(* IEC 61131-3 sources: plc_path_sender/, 1 file *)

(* ---- A1_Input_Normalizer.st ---- *)
(*****************************************************
 A1 Input Normalizer - ST Program Skeleton
 Purpose: Provide structure only; logic intentionally omitted.
*****************************************************)

PROGRAM A1_Input_Normalizer
VAR
    (* === Inputs from upstream sources === *)
    RawInput_1 : INT; (* Placeholder for raw input channel 1 *)
    RawInput_2 : INT; (* Placeholder for raw input channel 2 *)

    (* === Configuration / tuning parameters === *)
    ScaleFactor_1 : REAL; (* Placeholder for scaling factor *)
    Offset_1      : REAL; (* Placeholder for offset value *)

    (* === Internal state / intermediate values === *)
    Normalized_1 : REAL; (* Placeholder for normalized result *)
    Normalized_2 : REAL; (* Placeholder for normalized result *)

    (* === Outputs to downstream modules === *)
    Out_1 : REAL; (* Placeholder output channel 1 *)
    Out_2 : REAL; (* Placeholder output channel 2 *)
END_VAR

(* ---------------------------------------------------
   Section: Input acquisition
   Purpose: Read and buffer raw inputs for normalization.
--------------------------------------------------- *)
(* TODO: Insert input acquisition logic here. *)

(* ---------------------------------------------------
   Section: Range validation
   Purpose: Validate raw inputs and handle out-of-range cases.
--------------------------------------------------- *)
(* TODO: Insert range validation logic here. *)

(* ---------------------------------------------------
   Section: Normalization
   Purpose: Convert raw inputs into normalized values.
--------------------------------------------------- *)
(* TODO: Insert normalization logic here. *)

(* ---------------------------------------------------
   Section: Output assignment
   Purpose: Map normalized values to outputs for downstream use.
--------------------------------------------------- *)
(* TODO: Insert output assignment logic here. *)

END_PROGRAM
